   AI_710B.RAW_MIN := -2000;
   AI_710B.RAW_MAX := 8500;
   AI_710B.RAW_NAME := 'Thermal Resistance - 4-wire (Pt200 standard - 3916)';
   AI_710B.___________0030_1 := false;
   AI_710B.___________0030_2 := false;
   AI_710B.PARAM_TYPE := 16#07;
   AI_710B.PARAM_RANGE := 16#0B;
   AI_710B.PARAM_COEF := 16#01;
   AI_710B.VALUE_COEF := 0.003916;
   AI_730B.AI_CODE := 16#730B;
   AI_730B.___________0020_0 := false;
   AI_730B.___________0010_2 := false;
   AI_730B.RAW_MIN := -2000;
   AI_730B.RAW_MAX := 8500;
   AI_730B.RAW_NAME := 'Thermal Resistance - 4-wire (Pt200 standard - 392)';
   AI_730B.___________0030_1 := false;
   AI_730B.___________0030_2 := false;
   AI_730B.PARAM_TYPE := 16#07;
   AI_730B.PARAM_RANGE := 16#0B;
   AI_730B.PARAM_COEF := 16#03;
   AI_730B.VALUE_COEF := 0.00392;
   AI_7008.AI_CODE := 16#7008;
   AI_7008.___________0020_0 := false;
   AI_7008.___________0010_2 := false;
   AI_7008.RAW_MIN := -12000;
   AI_7008.RAW_MAX := 13000;
   AI_7008.RAW_NAME := 'Thermal Resistance - 4-wire (Pt500 climate - 3851)';
   AI_7008.___________0030_1 := false;
   AI_7008.___________0030_2 := false;
   AI_7008.PARAM_TYPE := 16#07;
   AI_7008.PARAM_RANGE := 16#08;
   AI_7008.PARAM_COEF := 16#00;
   AI_7008.VALUE_COEF := 0.003851;
   AI_7208.AI_CODE := 16#7208;
   AI_7208.___________0020_0 := false;
   AI_7208.___________0010_2 := false;
   AI_7208.RAW_MIN := -12000;
   AI_7208.RAW_MAX := 13000;
   AI_7208.RAW_NAME := 'Thermal Resistance - 4-wire (Pt500 climate - 3902)';
   AI_7208.___________0030_1 := false;
   AI_7208.___________0030_2 := false;
   AI_7208.PARAM_TYPE := 16#07;
   AI_7208.PARAM_RANGE := 16#08;
   AI_7208.PARAM_COEF := 16#02;
   AI_7208.VALUE_COEF := 0.003902;
   AI_7508.AI_CODE := 16#7508;
   AI_7508.___________0020_0 := false;
   AI_7508.___________0010_2 := false;
   AI_7508.RAW_MIN := -12000;
   AI_7508.RAW_MAX := 13000;
   AI_7508.RAW_NAME := 'Thermal Resistance - 4-wire (Pt500 climate - 391)';
   AI_7508.___________0030_1 := false;
   AI_7508.___________0030_2 := false;
   AI_7508.PARAM_TYPE := 16#07;
   AI_7508.PARAM_RANGE := 16#08;
   AI_7508.PARAM_COEF := 16#05;
   AI_7508.VALUE_COEF := 0.00391;
   AI_7108.AI_CODE := 16#7108;
   AI_7108.___________0020_0 := false;
   AI_7108.___________0010_2 := false;
   AI_7108.RAW_MIN := -12000;
   AI_7108.RAW_MAX := 13000;
   AI_7108.RAW_NAME := 'Thermal Resistance - 4-wire (Pt500 climate - 3916)';
   AI_7108.___________0030_1 := false;
   AI_7108.___________0030_2 := false;
   AI_7108.PARAM_TYPE := 16#07;
   AI_7108.PARAM_RANGE := 16#08;
   AI_7108.PARAM_COEF := 16#01;
   AI_7108.VALUE_COEF := 0.003916;
   AI_7308.AI_CODE := 16#7308;
   AI_7308.___________0020_0 := false;
   AI_7308.___________0010_2 := false;
   AI_7308.RAW_MIN := -12000;
   AI_7308.RAW_MAX := 13000;
   AI_7308.RAW_NAME := 'Thermal Resistance - 4-wire (Pt500 climate - 392)';
   AI_7308.___________0030_1 := false;
   AI_7308.___________0030_2 := false;
   AI_7308.PARAM_TYPE := 16#07;
   AI_7308.PARAM_RANGE := 16#08;
   AI_7308.PARAM_COEF := 16#03;
   AI_7308.VALUE_COEF := 0.00392;
   AI_7004.AI_CODE := 16#7004;
   AI_7004.___________0020_0 := false;
   AI_7004.___________0010_2 := false;
   AI_7004.RAW_MIN := -2000;
   AI_7004.RAW_MAX := 8500;
   AI_7004.RAW_NAME := 'Thermal Resistance - 4-wire (Pt500 standard - 3851)';
   AI_7004.___________0030_1 := false;
   AI_7004.___________0030_2 := false;
   AI_7004.PARAM_TYPE := 16#07;
   AI_7004.PARAM_RANGE := 16#04;
   AI_7004.PARAM_COEF := 16#00;
   AI_7004.VALUE_COEF := 0.003851;
   AI_7204.AI_CODE := 16#7204;
   AI_7204.___________0020_0 := false;
   AI_7204.___________0010_2 := false;
   AI_7204.RAW_MIN := -2000;
   AI_7204.RAW_MAX := 8500;
   AI_7204.RAW_NAME := 'Thermal Resistance - 4-wire (Pt500 standard - 3902)';
   AI_7204.___________0030_1 := false;
   AI_7204.___________0030_2 := false;
   AI_7204.PARAM_TYPE := 16#07;
   AI_7204.PARAM_RANGE := 16#04;
   AI_7204.PARAM_COEF := 16#02;
   AI_7204.VALUE_COEF := 0.003902;
   AI_7504.AI_CODE := 16#7504;
   AI_7504.___________0020_0 := false;
   AI_7504.___________0010_2 := false;
   AI_7504.RAW_MIN := -2000;
   AI_7504.RAW_MAX := 8500;
   AI_7504.RAW_NAME := 'Thermal Resistance - 4-wire (Pt500 standard - 391)';
   AI_7504.___________0030_1 := false;
   AI_7504.___________0030_2 := false;
   AI_7504.PARAM_TYPE := 16#07;
   AI_7504.PARAM_RANGE := 16#04;
   AI_7504.PARAM_COEF := 16#05;
   AI_7504.VALUE_COEF := 0.00391;
   AI_7104.AI_CODE := 16#7104;
   AI_7104.___________0020_0 := false;
   AI_7104.___________0010_2 := false;
   AI_7104.RAW_MIN := -2000;
   AI_7104.RAW_MAX := 8500;
   AI_7104.RAW_NAME := 'Thermal Resistance - 4-wire (Pt500 standard - 3916)';
   AI_7104.___________0030_1 := false;
   AI_7104.___________0030_2 := false;
   AI_7104.PARAM_TYPE := 16#07;
   AI_7104.PARAM_RANGE := 16#04;
   AI_7104.PARAM_COEF := 16#01;
   AI_7104.VALUE_COEF := 0.003916;
   AI_7304.AI_CODE := 16#7304;
   AI_7304.___________0020_0 := false;
   AI_7304.___________0010_2 := false;
   AI_7304.RAW_MIN := -2000;
   AI_7304.RAW_MAX := 8500;
   AI_7304.RAW_NAME := 'Thermal Resistance - 4-wire (Pt500 standard - 392)';
   AI_7304.___________0030_1 := false;
   AI_7304.___________0030_2 := false;
   AI_7304.PARAM_TYPE := 16#07;
   AI_7304.PARAM_RANGE := 16#04;
   AI_7304.PARAM_COEF := 16#03;
   AI_7304.VALUE_COEF := 0.00392;
   AI_7009.AI_CODE := 16#7009;
   AI_7009.___________0020_0 := false;
   AI_7009.___________0010_2 := false;
   AI_7009.RAW_MIN := -12000;
   AI_7009.RAW_MAX := 13000;
   AI_7009.RAW_NAME := 'Thermal Resistance - 4-wire (Pt1000 climate - 3851)';
   AI_7009.___________0030_1 := false;
   AI_7009.___________0030_2 := false;
   AI_7009.PARAM_TYPE := 16#07;
   AI_7009.PARAM_RANGE := 16#09;
   AI_7009.PARAM_COEF := 16#00;
   AI_7009.VALUE_COEF := 0.003851;
   AI_7209.AI_CODE := 16#7209;
   AI_7209.___________0020_0 := false;
   AI_7209.___________0010_2 := false;
   AI_7209.RAW_MIN := -12000;
   AI_7209.RAW_MAX := 13000;
   AI_7209.RAW_NAME := 'Thermal Resistance - 4-wire (Pt1000 climate - 3902)';
   AI_7209.___________0030_1 := false;
   AI_7209.___________0030_2 := false;
   AI_7209.PARAM_TYPE := 16#07;
   AI_7209.PARAM_RANGE := 16#09;
   AI_7209.PARAM_COEF := 16#02;
   AI_7209.VALUE_COEF := 0.003902;
   AI_7509.AI_CODE := 16#7509;
   AI_7509.___________0020_0 := false;
   AI_7509.___________0010_2 := false;
   AI_7509.RAW_MIN := -12000;
   AI_7509.RAW_MAX := 13000;
   AI_7509.RAW_NAME := 'Thermal Resistance - 4-wire (Pt1000 climate - 391)';
   AI_7509.___________0030_1 := false;
   AI_7509.___________0030_2 := false;
   AI_7509.PARAM_TYPE := 16#07;
   AI_7509.PARAM_RANGE := 16#09;
   AI_7509.PARAM_COEF := 16#05;
   AI_7509.VALUE_COEF := 0.00391;
   AI_7109.AI_CODE := 16#7109;
   AI_7109.___________0020_0 := false;
   AI_7109.___________0010_2 := false;
   AI_7109.RAW_MIN := -12000;
   AI_7109.RAW_MAX := 13000;
   AI_7109.RAW_NAME := 'Thermal Resistance - 4-wire (Pt1000 climate - 3916)';
   AI_7109.___________0030_1 := false;
   AI_7109.___________0030_2 := false;
   AI_7109.PARAM_TYPE := 16#07;
   AI_7109.PARAM_RANGE := 16#09;
   AI_7109.PARAM_COEF := 16#01;
   AI_7109.VALUE_COEF := 0.003916;
   AI_7309.AI_CODE := 16#7309;
   AI_7309.___________0020_0 := false;
   AI_7309.___________0010_2 := false;
   AI_7309.RAW_MIN := -12000;
   AI_7309.RAW_MAX := 13000;
   AI_7309.RAW_NAME := 'Thermal Resistance - 4-wire (Pt1000 climate - 392)';
   AI_7309.___________0030_1 := false;
   AI_7309.___________0030_2 := false;
   AI_7309.PARAM_TYPE := 16#07;
   AI_7309.PARAM_RANGE := 16#09;
   AI_7309.PARAM_COEF := 16#03;
   AI_7309.VALUE_COEF := 0.00392;
   AI_7005.AI_CODE := 16#7005;
   AI_7005.___________0020_0 := false;
   AI_7005.___________0010_2 := false;
   AI_7005.RAW_MIN := -2000;
   AI_7005.RAW_MAX := 8500;
   AI_7005.RAW_NAME := 'Thermal Resistance - 4-wire (Pt1000 standard - 3851)';
   AI_7005.___________0030_1 := false;
   AI_7005.___________0030_2 := false;
   AI_7005.PARAM_TYPE := 16#07;
   AI_7005.PARAM_RANGE := 16#05;
   AI_7005.PARAM_COEF := 16#00;
   AI_7005.VALUE_COEF := 0.003851;
   AI_7205.AI_CODE := 16#7205;
   AI_7205.___________0020_0 := false;
   AI_7205.___________0010_2 := false;
   AI_7205.RAW_MIN := -2000;
   AI_7205.RAW_MAX := 8500;
   AI_7205.RAW_NAME := 'Thermal Resistance - 4-wire (Pt1000 standard - 3902)';
   AI_7205.___________0030_1 := false;
   AI_7205.___________0030_2 := false;
   AI_7205.PARAM_TYPE := 16#07;
   AI_7205.PARAM_RANGE := 16#05;
   AI_7205.PARAM_COEF := 16#02;
   AI_7205.VALUE_COEF := 0.003902;
   AI_7505.AI_CODE := 16#7505;
   AI_7505.___________0020_0 := false;
   AI_7505.___________0010_2 := false;
   AI_7505.RAW_MIN := -2000;
   AI_7505.RAW_MAX := 8500;
   AI_7505.RAW_NAME := 'Thermal Resistance - 4-wire (Pt1000 standard - 391)';
   AI_7505.___________0030_1 := false;
   AI_7505.___________0030_2 := false;
   AI_7505.PARAM_TYPE := 16#07;
   AI_7505.PARAM_RANGE := 16#05;
   AI_7505.PARAM_COEF := 16#05;
   AI_7505.VALUE_COEF := 0.00391;
   AI_7105.AI_CODE := 16#7105;
   AI_7105.___________0020_0 := false;
   AI_7105.___________0010_2 := false;
   AI_7105.RAW_MIN := -2000;
   AI_7105.RAW_MAX := 8500;
   AI_7105.RAW_NAME := 'Thermal Resistance - 4-wire (Pt1000 standard - 3916)';
   AI_7105.___________0030_1 := false;
   AI_7105.___________0030_2 := false;
   AI_7105.PARAM_TYPE := 16#07;
   AI_7105.PARAM_RANGE := 16#05;
   AI_7105.PARAM_COEF := 16#01;
   AI_7105.VALUE_COEF := 0.003916;
   AI_7305.AI_CODE := 16#7305;
   AI_7305.___________0020_0 := false;
   AI_7305.___________0010_2 := false;
   AI_7305.RAW_MIN := -2000;
   AI_7305.RAW_MAX := 8500;
   AI_7305.RAW_NAME := 'Thermal Resistance - 4-wire (Pt1000 standard - 392)';
   AI_7305.___________0030_1 := false;
   AI_7305.___________0030_2 := false;
   AI_7305.PARAM_TYPE := 16#07;
   AI_7305.PARAM_RANGE := 16#05;
   AI_7305.PARAM_COEF := 16#03;
   AI_7305.VALUE_COEF := 0.00392;
   AI_8B0E.AI_CODE := 16#8B0E;
   AI_8B0E.___________0020_0 := false;
   AI_8B0E.___________0010_2 := false;
   AI_8B0E.RAW_MIN := -5000;
   AI_8B0E.RAW_MAX := 15000;
   AI_8B0E.RAW_NAME := 'Thermal Resistance - 3-wire (Cu10 climate - 426)';
   AI_8B0E.___________0030_1 := false;
   AI_8B0E.___________0030_2 := false;
   AI_8B0E.PARAM_TYPE := 16#08;
   AI_8B0E.PARAM_RANGE := 16#0E;
   AI_8B0E.PARAM_COEF := 16#0B;
   AI_8B0E.VALUE_COEF := 0.00426;
   AI_8C0E.AI_CODE := 16#8C0E;
   AI_8C0E.___________0020_0 := false;
   AI_8C0E.___________0010_2 := false;
   AI_8C0E.RAW_MIN := -5000;
   AI_8C0E.RAW_MAX := 15000;
   AI_8C0E.RAW_NAME := 'Thermal Resistance - 3-wire (Cu10 climate - 427)';
   AI_8C0E.___________0030_1 := false;
   AI_8C0E.___________0030_2 := false;
   AI_8C0E.PARAM_TYPE := 16#08;
   AI_8C0E.PARAM_RANGE := 16#0E;
   AI_8C0E.PARAM_COEF := 16#0C;
   AI_8C0E.VALUE_COEF := 0.00427;
   AI_8D0E.AI_CODE := 16#8D0E;
   AI_8D0E.___________0020_0 := false;
   AI_8D0E.___________0010_2 := false;
   AI_8D0E.RAW_MIN := -5000;
   AI_8D0E.RAW_MAX := 15000;
   AI_8D0E.RAW_NAME := 'Thermal Resistance - 3-wire (Cu10 climate - 428)';
   AI_8D0E.___________0030_1 := false;
   AI_8D0E.___________0030_2 := false;
   AI_8D0E.PARAM_TYPE := 16#08;
   AI_8D0E.PARAM_RANGE := 16#0E;
   AI_8D0E.PARAM_COEF := 16#0D;
   AI_8D0E.VALUE_COEF := 0.00428;
   AI_8B0F.AI_CODE := 16#8B0F;
   AI_8B0F.___________0020_0 := false;
   AI_8B0F.___________0010_2 := false;
   AI_8B0F.RAW_MIN := -500;
   AI_8B0F.RAW_MAX := 2000;
   AI_8B0F.RAW_NAME := 'Thermal Resistance - 3-wire (Cu10 standard - 426)';
   AI_8B0F.___________0030_1 := false;
   AI_8B0F.___________0030_2 := false;
   AI_8B0F.PARAM_TYPE := 16#08;
   AI_8B0F.PARAM_RANGE := 16#0F;
   AI_8B0F.PARAM_COEF := 16#0B;
   AI_8B0F.VALUE_COEF := 0.00426;
   AI_8C0F.AI_CODE := 16#8C0F;
   AI_8C0F.___________0020_0 := false;
   AI_8C0F.___________0010_2 := false;
   AI_8C0F.RAW_MIN := -2000;
   AI_8C0F.RAW_MAX := 2600;
   AI_8C0F.RAW_NAME := 'Thermal Resistance - 3-wire (Cu10 standard - 427)';
   AI_8C0F.___________0030_1 := false;
   AI_8C0F.___________0030_2 := false;
   AI_8C0F.PARAM_TYPE := 16#08;
   AI_8C0F.PARAM_RANGE := 16#0F;
   AI_8C0F.PARAM_COEF := 16#0C;
   AI_8C0F.VALUE_COEF := 0.00427;
   AI_8D0F.AI_CODE := 16#8D0F;
   AI_8D0F.___________0020_0 := false;
   AI_8D0F.___________0010_2 := false;
   AI_8D0F.RAW_MIN := -1800;
   AI_8D0F.RAW_MAX := 2000;
   AI_8D0F.RAW_NAME := 'Thermal Resistance - 3-wire (Cu10 standard - 428)';
   AI_8D0F.___________0030_1 := false;
   AI_8D0F.___________0030_2 := false;
   AI_8D0F.PARAM_TYPE := 16#08;
   AI_8D0F.PARAM_RANGE := 16#0F;
   AI_8D0F.PARAM_COEF := 16#0D;
   AI_8D0F.VALUE_COEF := 0.00428;
   AI_8B19.AI_CODE := 16#8B19;
   AI_8B19.___________0020_0 := false;
   AI_8B19.___________0010_2 := false;
   AI_8B19.RAW_MIN := -5000;
   AI_8B19.RAW_MAX := 15000;
   AI_8B19.RAW_NAME := 'Thermal Resistance - 3-wire (Cu50 climate - 426)';
   AI_8B19.___________0030_1 := false;
   AI_8B19.___________0030_2 := false;
   AI_8B19.PARAM_TYPE := 16#08;
   AI_8B19.PARAM_RANGE := 16#19;
   AI_8B19.PARAM_COEF := 16#0B;
   AI_8B19.VALUE_COEF := 0.00426;
   AI_8C19.AI_CODE := 16#8C19;
   AI_8C19.___________0020_0 := false;
   AI_8C19.___________0010_2 := false;
   AI_8C19.RAW_MIN := -5000;
   AI_8C19.RAW_MAX := 15000;
   AI_8C19.RAW_NAME := 'Thermal Resistance - 3-wire (Cu50 climate - 427)';
   AI_8C19.___________0030_1 := false;
   AI_8C19.___________0030_2 := false;
   AI_8C19.PARAM_TYPE := 16#08;
   AI_8C19.PARAM_RANGE := 16#19;
   AI_8C19.PARAM_COEF := 16#0C;
   AI_8C19.VALUE_COEF := 0.00427;
   AI_8D19.AI_CODE := 16#8D19;
   AI_8D19.___________0020_0 := false;
   AI_8D19.___________0010_2 := false;
   AI_8D19.RAW_MIN := -5000;
   AI_8D19.RAW_MAX := 15000;
   AI_8D19.RAW_NAME := 'Thermal Resistance - 3-wire (Cu50 climate - 428)';
   AI_8D19.___________0030_1 := false;
   AI_8D19.___________0030_2 := false;
   AI_8D19.PARAM_TYPE := 16#08;
   AI_8D19.PARAM_RANGE := 16#19;
   AI_8D19.PARAM_COEF := 16#0D;
   AI_8D19.VALUE_COEF := 0.00428;
   AI_8B18.AI_CODE := 16#8B18;
   AI_8B18.___________0020_0 := false;
   AI_8B18.___________0010_2 := false;
   AI_8B18.RAW_MIN := -500;
   AI_8B18.RAW_MAX := 2000;
   AI_8B18.RAW_NAME := 'Thermal Resistance - 3-wire (Cu50 standard - 426)';
   AI_8B18.___________0030_1 := false;
   AI_8B18.___________0030_2 := false;
   AI_8B18.PARAM_TYPE := 16#08;
   AI_8B18.PARAM_RANGE := 16#18;
   AI_8B18.PARAM_COEF := 16#0B;
   AI_8B18.VALUE_COEF := 0.00426;
   AI_8C18.AI_CODE := 16#8C18;
   AI_8C18.___________0020_0 := false;
   AI_8C18.___________0010_2 := false;
   AI_8C18.RAW_MIN := -2000;
   AI_8C18.RAW_MAX := 2600;
   AI_8C18.RAW_NAME := 'Thermal Resistance - 3-wire (Cu50 standard - 427)';
   AI_8C18.___________0030_1 := false;
   AI_8C18.___________0030_2 := false;
   AI_8C18.PARAM_TYPE := 16#08;
   AI_8C18.PARAM_RANGE := 16#18;
   AI_8C18.PARAM_COEF := 16#0C;
   AI_8C18.VALUE_COEF := 0.00427;
   AI_8D18.AI_CODE := 16#8D18;
   AI_8D18.___________0020_0 := false;
   AI_8D18.___________0010_2 := false;
   AI_8D18.RAW_MIN := -1800;
   AI_8D18.RAW_MAX := 2000;
   AI_8D18.RAW_NAME := 'Thermal Resistance - 3-wire (Cu50 standard - 428)';
   AI_8D18.___________0030_1 := false;
   AI_8D18.___________0030_2 := false;
   AI_8D18.PARAM_TYPE := 16#08;
   AI_8D18.PARAM_RANGE := 16#18;
   AI_8D18.PARAM_COEF := 16#0D;
   AI_8D18.VALUE_COEF := 0.00428;
   AI_8B1B.AI_CODE := 16#8B1B;
   AI_8B1B.___________0020_0 := false;
   AI_8B1B.___________0010_2 := false;
   AI_8B1B.RAW_MIN := -5000;
   AI_8B1B.RAW_MAX := 15000;
   AI_8B1B.RAW_NAME := 'Thermal Resistance - 3-wire (Cu100 climate - 426)';
   AI_8B1B.___________0030_1 := false;
   AI_8B1B.___________0030_2 := false;
   AI_8B1B.PARAM_TYPE := 16#08;
   AI_8B1B.PARAM_RANGE := 16#1B;
   AI_8B1B.PARAM_COEF := 16#0B;
   AI_8B1B.VALUE_COEF := 0.00426;
   AI_8C1B.AI_CODE := 16#8C1B;
   AI_8C1B.___________0020_0 := false;
   AI_8C1B.___________0010_2 := false;
   AI_8C1B.RAW_MIN := -5000;
   AI_8C1B.RAW_MAX := 15000;
   AI_8C1B.RAW_NAME := 'Thermal Resistance - 3-wire (Cu100 climate - 427)';
   AI_8C1B.___________0030_1 := false;
   AI_8C1B.___________0030_2 := false;
   AI_8C1B.PARAM_TYPE := 16#08;
   AI_8C1B.PARAM_RANGE := 16#1B;
   AI_8C1B.PARAM_COEF := 16#0C;
   AI_8C1B.VALUE_COEF := 0.00427;
   AI_8D1B.AI_CODE := 16#8D1B;
   AI_8D1B.___________0020_0 := false;
   AI_8D1B.___________0010_2 := false;
   AI_8D1B.RAW_MIN := -5000;
   AI_8D1B.RAW_MAX := 15000;
   AI_8D1B.RAW_NAME := 'Thermal Resistance - 3-wire (Cu100 climate - 428)';
   AI_8D1B.___________0030_1 := false;
   AI_8D1B.___________0030_2 := false;
   AI_8D1B.PARAM_TYPE := 16#08;
   AI_8D1B.PARAM_RANGE := 16#1B;
   AI_8D1B.PARAM_COEF := 16#0D;
   AI_8D1B.VALUE_COEF := 0.00428;
   AI_8B1A.AI_CODE := 16#8B1A;
   AI_8B1A.___________0020_0 := false;
   AI_8B1A.___________0010_2 := false;
   AI_8B1A.RAW_MIN := -500;
   AI_8B1A.RAW_MAX := 2000;
   AI_8B1A.RAW_NAME := 'Thermal Resistance - 3-wire (Cu100 standard - 426)';
   AI_8B1A.___________0030_1 := false;
   AI_8B1A.___________0030_2 := false;
   AI_8B1A.PARAM_TYPE := 16#08;
   AI_8B1A.PARAM_RANGE := 16#1A;
   AI_8B1A.PARAM_COEF := 16#0B;
   AI_8B1A.VALUE_COEF := 0.00426;
   AI_8C1A.AI_CODE := 16#8C1A;
   AI_8C1A.___________0020_0 := false;
   AI_8C1A.___________0010_2 := false;
   AI_8C1A.RAW_MIN := -2000;
   AI_8C1A.RAW_MAX := 2600;
   AI_8C1A.RAW_NAME := 'Thermal Resistance - 3-wire (Cu100 standard - 427)';
   AI_8C1A.___________0030_1 := false;
   AI_8C1A.___________0030_2 := false;
   AI_8C1A.PARAM_TYPE := 16#08;
   AI_8C1A.PARAM_RANGE := 16#1A;
   AI_8C1A.PARAM_COEF := 16#0C;
   AI_8C1A.VALUE_COEF := 0.00427;
   AI_8D1A.AI_CODE := 16#8D1A;
   AI_8D1A.___________0020_0 := false;
   AI_8D1A.___________0010_2 := false;
   AI_8D1A.RAW_MIN := -1800;
   AI_8D1A.RAW_MAX := 2000;
   AI_8D1A.RAW_NAME := 'Thermal Resistance - 3-wire (Cu100 standard - 428)';
   AI_8D1A.___________0030_1 := false;
   AI_8D1A.___________0030_2 := false;
   AI_8D1A.PARAM_TYPE := 16#08;
   AI_8D1A.PARAM_RANGE := 16#1A;
   AI_8D1A.PARAM_COEF := 16#0D;
   AI_8D1A.VALUE_COEF := 0.00428;
   AI_8A1D.AI_CODE := 16#8A1D;
   AI_8A1D.___________0020_0 := false;
   AI_8A1D.___________0010_2 := false;
   AI_8A1D.RAW_MIN := -6000;
   AI_8A1D.RAW_MAX := 13000;
   AI_8A1D.RAW_NAME := 'Thermal Resistance - 3-wire (LG-Ni1000 climate - 500)';
   AI_8A1D.___________0030_1 := false;
   AI_8A1D.___________0030_2 := false;
   AI_8A1D.PARAM_TYPE := 16#08;
   AI_8A1D.PARAM_RANGE := 16#1D;
   AI_8A1D.PARAM_COEF := 16#0A;
   AI_8A1D.VALUE_COEF := 0.005;
   AI_8A1C.AI_CODE := 16#8A1C;
   AI_8A1C.___________0020_0 := false;
   AI_8A1C.___________0010_2 := false;
   AI_8A1C.RAW_MIN := -600;
   AI_8A1C.RAW_MAX := 2500;
   AI_8A1C.RAW_NAME := 'Thermal Resistance - 3-wire (LG-Ni1000 standard - 500)';
   AI_8A1C.___________0030_1 := false;
   AI_8A1C.___________0030_2 := false;
   AI_8A1C.PARAM_TYPE := 16#08;
   AI_8A1C.PARAM_RANGE := 16#1C;
   AI_8A1C.PARAM_COEF := 16#0A;
   AI_8A1C.VALUE_COEF := 0.005;
   AI_871F.AI_CODE := 16#871F;
   AI_871F.___________0020_0 := false;
   AI_871F.___________0010_2 := false;
   AI_871F.RAW_MIN := -6000;
   AI_871F.RAW_MAX := 13000;
   AI_871F.RAW_NAME := 'Thermal Resistance - 3-wire (Ni10 climate - 617)';
   AI_871F.___________0030_1 := false;
   AI_871F.___________0030_2 := false;
   AI_871F.PARAM_TYPE := 16#08;
   AI_871F.PARAM_RANGE := 16#1F;
   AI_871F.PARAM_COEF := 16#07;
   AI_871F.VALUE_COEF := 0.00617;
   AI_881F.AI_CODE := 16#881F;
   AI_881F.___________0020_0 := false;
   AI_881F.___________0010_2 := false;
   AI_881F.RAW_MIN := -6000;
   AI_881F.RAW_MAX := 13000;
   AI_881F.RAW_NAME := 'Thermal Resistance - 3-wire (Ni10 climate - 618)';
   AI_881F.___________0030_1 := false;
   AI_881F.___________0030_2 := false;
   AI_881F.PARAM_TYPE := 16#08;
   AI_881F.PARAM_RANGE := 16#1F;
   AI_881F.PARAM_COEF := 16#08;
   AI_881F.VALUE_COEF := 0.00618;
   AI_891F.AI_CODE := 16#891F;
   AI_891F.___________0020_0 := false;
   AI_891F.___________0010_2 := false;
   AI_891F.RAW_MIN := -6000;
   AI_891F.RAW_MAX := 13000;
   AI_891F.RAW_NAME := 'Thermal Resistance - 3-wire (Ni10 climate - 672)';
   AI_891F.___________0030_1 := false;
   AI_891F.___________0030_2 := false;
   AI_891F.PARAM_TYPE := 16#08;
   AI_891F.PARAM_RANGE := 16#1F;
   AI_891F.PARAM_COEF := 16#09;
   AI_891F.VALUE_COEF := 0.00672;
   AI_871E.AI_CODE := 16#871E;
   AI_871E.___________0020_0 := false;
   AI_871E.___________0010_2 := false;
   AI_871E.RAW_MIN := -600;
   AI_871E.RAW_MAX := 1800;
   AI_871E.RAW_NAME := 'Thermal Resistance - 3-wire (Ni10 standard - 617)';
   AI_871E.___________0030_1 := false;
   AI_871E.___________0030_2 := false;
   AI_871E.PARAM_TYPE := 16#08;
   AI_871E.PARAM_RANGE := 16#1E;
   AI_871E.PARAM_COEF := 16#07;
   AI_871E.VALUE_COEF := 0.00617;
   AI_881E.AI_CODE := 16#881E;
   AI_881E.___________0020_0 := false;
   AI_881E.___________0010_2 := false;
   AI_881E.RAW_MIN := -600;
   AI_881E.RAW_MAX := 2500;
   AI_881E.RAW_NAME := 'Thermal Resistance - 3-wire (Ni10 standard - 618)';
   AI_881E.___________0030_1 := false;
   AI_881E.___________0030_2 := false;
   AI_881E.PARAM_TYPE := 16#08;
   AI_881E.PARAM_RANGE := 16#1E;
   AI_881E.PARAM_COEF := 16#08;
   AI_881E.VALUE_COEF := 0.00618;
   AI_891E.AI_CODE := 16#891E;
   AI_891E.___________0020_0 := false;
   AI_891E.___________0010_2 := false;
   AI_891E.RAW_MIN := -600;
   AI_891E.RAW_MAX := 2500;
   AI_891E.RAW_NAME := 'Thermal Resistance - 3-wire (Ni10 standard - 672)';
   AI_891E.___________0030_1 := false;
   AI_891E.___________0030_2 := false;
   AI_891E.PARAM_TYPE := 16#08;
   AI_891E.PARAM_RANGE := 16#1E;
   AI_891E.PARAM_COEF := 16#09;
   AI_891E.VALUE_COEF := 0.00672;
   AI_870D.AI_CODE := 16#870D;
   AI_870D.___________0020_0 := false;
   AI_870D.___________0010_2 := false;
   AI_870D.RAW_MIN := -6000;
   AI_870D.RAW_MAX := 13000;
   AI_870D.RAW_NAME := 'Thermal Resistance - 3-wire (Ni120 climate - 617)';
   AI_870D.___________0030_1 := false;
   AI_870D.___________0030_2 := false;
   AI_870D.PARAM_TYPE := 16#08;
   AI_870D.PARAM_RANGE := 16#0D;
   AI_870D.PARAM_COEF := 16#07;
   AI_870D.VALUE_COEF := 0.00617;
   AI_880D.AI_CODE := 16#880D;
   AI_880D.___________0020_0 := false;
   AI_880D.___________0010_2 := false;
   AI_880D.RAW_MIN := -6000;
   AI_880D.RAW_MAX := 13000;
   AI_880D.RAW_NAME := 'Thermal Resistance - 3-wire (Ni120 climate - 618)';
   AI_880D.___________0030_1 := false;
   AI_880D.___________0030_2 := false;
   AI_880D.PARAM_TYPE := 16#08;
   AI_880D.PARAM_RANGE := 16#0D;
   AI_880D.PARAM_COEF := 16#08;
   AI_880D.VALUE_COEF := 0.00618;
   AI_890D.AI_CODE := 16#890D;
   AI_890D.___________0020_0 := false;
   AI_890D.___________0010_2 := false;
   AI_890D.RAW_MIN := -6000;
   AI_890D.RAW_MAX := 13000;
   AI_890D.RAW_NAME := 'Thermal Resistance - 3-wire (Ni120 climate - 672)';
   AI_890D.___________0030_1 := false;
   AI_890D.___________0030_2 := false;
   AI_890D.PARAM_TYPE := 16#08;
   AI_890D.PARAM_RANGE := 16#0D;
   AI_890D.PARAM_COEF := 16#09;
   AI_890D.VALUE_COEF := 0.00672;
   AI_870C.AI_CODE := 16#870C;
   AI_870C.___________0020_0 := false;
   AI_870C.___________0010_2 := false;
   AI_870C.RAW_MIN := -600;
   AI_870C.RAW_MAX := 1800;
   AI_870C.RAW_NAME := 'Thermal Resistance - 3-wire (Ni120 standard - 617)';
   AI_870C.___________0030_1 := false;
   AI_870C.___________0030_2 := false;
   AI_870C.PARAM_TYPE := 16#08;
   AI_870C.PARAM_RANGE := 16#0C;
   AI_870C.PARAM_COEF := 16#07;
   AI_870C.VALUE_COEF := 0.00617;
   AI_880C.AI_CODE := 16#880C;
   AI_880C.___________0020_0 := false;
   AI_880C.___________0010_2 := false;
   AI_880C.RAW_MIN := -600;
   AI_880C.RAW_MAX := 2500;
   AI_880C.RAW_NAME := 'Thermal Resistance - 3-wire (Ni120 standard - 618)';
   AI_880C.___________0030_1 := false;
   AI_880C.___________0030_2 := false;
   AI_880C.PARAM_TYPE := 16#08;
   AI_880C.PARAM_RANGE := 16#0C;
   AI_880C.PARAM_COEF := 16#08;
   AI_880C.VALUE_COEF := 0.00618;
   AI_890C.AI_CODE := 16#890C;
   AI_890C.___________0020_0 := false;
   AI_890C.___________0010_2 := false;
   AI_890C.RAW_MIN := -600;
   AI_890C.RAW_MAX := 2500;
   AI_890C.RAW_NAME := 'Thermal Resistance - 3-wire (Ni120 standard - 672)';
   AI_890C.___________0030_1 := false;
   AI_890C.___________0030_2 := false;
   AI_890C.PARAM_TYPE := 16#08;
   AI_890C.PARAM_RANGE := 16#0C;
   AI_890C.PARAM_COEF := 16#09;
   AI_890C.VALUE_COEF := 0.00672;
   AI_8701.AI_CODE := 16#8701;
   AI_8701.___________0020_0 := false;
   AI_8701.___________0010_2 := false;
   AI_8701.RAW_MIN := -6000;
   AI_8701.RAW_MAX := 13000;
   AI_8701.RAW_NAME := 'Thermal Resistance - 3-wire (Ni100 climate - 617)';
   AI_8701.___________0030_1 := false;
   AI_8701.___________0030_2 := false;
   AI_8701.PARAM_TYPE := 16#08;
   AI_8701.PARAM_RANGE := 16#01;
   AI_8701.PARAM_COEF := 16#07;
   AI_8701.VALUE_COEF := 0.00617;
   AI_8801.AI_CODE := 16#8801;
   AI_8801.___________0020_0 := false;
   AI_8801.___________0010_2 := false;
   AI_8801.RAW_MIN := -6000;
   AI_8801.RAW_MAX := 13000;
   AI_8801.RAW_NAME := 'Thermal Resistance - 3-wire (Ni100 climate - 618)';
   AI_8801.___________0030_1 := false;
   AI_8801.___________0030_2 := false;
   AI_8801.PARAM_TYPE := 16#08;
   AI_8801.PARAM_RANGE := 16#01;
   AI_8801.PARAM_COEF := 16#08;
   AI_8801.VALUE_COEF := 0.00618;
   AI_8901.AI_CODE := 16#8901;
   AI_8901.___________0020_0 := false;
   AI_8901.___________0010_2 := false;
   AI_8901.RAW_MIN := -6000;
   AI_8901.RAW_MAX := 13000;
   AI_8901.RAW_NAME := 'Thermal Resistance - 3-wire (Ni100 climate - 672)';
   AI_8901.___________0030_1 := false;
   AI_8901.___________0030_2 := false;
   AI_8901.PARAM_TYPE := 16#08;
   AI_8901.PARAM_RANGE := 16#01;
   AI_8901.PARAM_COEF := 16#09;
   AI_8901.VALUE_COEF := 0.00672;
   AI_8703.AI_CODE := 16#8703;
   AI_8703.___________0020_0 := false;
   AI_8703.___________0010_2 := false;
   AI_8703.RAW_MIN := -600;
   AI_8703.RAW_MAX := 1800;
   AI_8703.RAW_NAME := 'Thermal Resistance - 3-wire (Ni100 standard - 617)';
   AI_8703.___________0030_1 := false;
   AI_8703.___________0030_2 := false;
   AI_8703.PARAM_TYPE := 16#08;
   AI_8703.PARAM_RANGE := 16#03;
   AI_8703.PARAM_COEF := 16#07;
   AI_8703.VALUE_COEF := 0.00617;
   AI_8803.AI_CODE := 16#8803;
   AI_8803.___________0020_0 := false;
   AI_8803.___________0010_2 := false;
   AI_8803.RAW_MIN := -600;
   AI_8803.RAW_MAX := 2500;
   AI_8803.RAW_NAME := 'Thermal Resistance - 3-wire (Ni100 standard - 618)';
   AI_8803.___________0030_1 := false;
   AI_8803.___________0030_2 := false;
   AI_8803.PARAM_TYPE := 16#08;
   AI_8803.PARAM_RANGE := 16#03;
   AI_8803.PARAM_COEF := 16#08;
   AI_8803.VALUE_COEF := 0.00618;
   AI_8903.AI_CODE := 16#8903;
   AI_8903.___________0020_0 := false;
   AI_8903.___________0010_2 := false;
   AI_8903.RAW_MIN := -600;
   AI_8903.RAW_MAX := 2500;
   AI_8903.RAW_NAME := 'Thermal Resistance - 3-wire (Ni100 standard - 672)';
   AI_8903.___________0030_1 := false;
   AI_8903.___________0030_2 := false;
   AI_8903.PARAM_TYPE := 16#08;
   AI_8903.PARAM_RANGE := 16#03;
   AI_8903.PARAM_COEF := 16#09;
   AI_8903.VALUE_COEF := 0.00672;
   AI_8711.AI_CODE := 16#8711;
   AI_8711.___________0020_0 := false;
   AI_8711.___________0010_2 := false;
   AI_8711.RAW_MIN := -6000;
   AI_8711.RAW_MAX := 13000;
   AI_8711.RAW_NAME := 'Thermal Resistance - 3-wire (Ni200 climate - 617)';
   AI_8711.___________0030_1 := false;
   AI_8711.___________0030_2 := false;
   AI_8711.PARAM_TYPE := 16#08;
   AI_8711.PARAM_RANGE := 16#11;
   AI_8711.PARAM_COEF := 16#07;
   AI_8711.VALUE_COEF := 0.00617;
   AI_8811.AI_CODE := 16#8811;
   AI_8811.___________0020_0 := false;
   AI_8811.___________0010_2 := false;
   AI_8811.RAW_MIN := -6000;
   AI_8811.RAW_MAX := 13000;
   AI_8811.RAW_NAME := 'Thermal Resistance - 3-wire (Ni200 climate - 618)';
   AI_8811.___________0030_1 := false;
   AI_8811.___________0030_2 := false;
   AI_8811.PARAM_TYPE := 16#08;
   AI_8811.PARAM_RANGE := 16#11;
   AI_8811.PARAM_COEF := 16#08;
   AI_8811.VALUE_COEF := 0.00618;
   AI_8911.AI_CODE := 16#8911;
   AI_8911.___________0020_0 := false;
   AI_8911.___________0010_2 := false;
   AI_8911.RAW_MIN := -6000;
   AI_8911.RAW_MAX := 13000;
   AI_8911.RAW_NAME := 'Thermal Resistance - 3-wire (Ni200 climate - 672)';
   AI_8911.___________0030_1 := false;
   AI_8911.___________0030_2 := false;
   AI_8911.PARAM_TYPE := 16#08;
   AI_8911.PARAM_RANGE := 16#11;
   AI_8911.PARAM_COEF := 16#09;
   AI_8911.VALUE_COEF := 0.00672;
   AI_8710.AI_CODE := 16#8710;
   AI_8710.___________0020_0 := false;
   AI_8710.___________0010_2 := false;
   AI_8710.RAW_MIN := -600;
   AI_8710.RAW_MAX := 1800;
   AI_8710.RAW_NAME := 'Thermal Resistance - 3-wire (Ni200 standard - 617)';
   AI_8710.___________0030_1 := false;
   AI_8710.___________0030_2 := false;
   AI_8710.PARAM_TYPE := 16#08;
   AI_8710.PARAM_RANGE := 16#10;
   AI_8710.PARAM_COEF := 16#07;
   AI_8710.VALUE_COEF := 0.00617;
   AI_8810.AI_CODE := 16#8810;
   AI_8810.___________0020_0 := false;
   AI_8810.___________0010_2 := false;
   AI_8810.RAW_MIN := -600;
   AI_8810.RAW_MAX := 2500;
   AI_8810.RAW_NAME := 'Thermal Resistance - 3-wire (Ni200 standard - 618)';
   AI_8810.___________0030_1 := false;
   AI_8810.___________0030_2 := false;
   AI_8810.PARAM_TYPE := 16#08;
   AI_8810.PARAM_RANGE := 16#10;
   AI_8810.PARAM_COEF := 16#08;
   AI_8810.VALUE_COEF := 0.00618;
   AI_8910.AI_CODE := 16#8910;
   AI_8910.___________0020_0 := false;
   AI_8910.___________0010_2 := false;
   AI_8910.RAW_MIN := -600;
   AI_8910.RAW_MAX := 2500;
   AI_8910.RAW_NAME := 'Thermal Resistance - 3-wire (Ni200 standard - 672)';
   AI_8910.___________0030_1 := false;
   AI_8910.___________0030_2 := false;
   AI_8910.PARAM_TYPE := 16#08;
   AI_8910.PARAM_RANGE := 16#10;
   AI_8910.PARAM_COEF := 16#09;
   AI_8910.VALUE_COEF := 0.00672;
   AI_8713.AI_CODE := 16#8713;
   AI_8713.___________0020_0 := false;
   AI_8713.___________0010_2 := false;
   AI_8713.RAW_MIN := -6000;
   AI_8713.RAW_MAX := 13000;
   AI_8713.RAW_NAME := 'Thermal Resistance - 3-wire (Ni500 climate - 617)';
   AI_8713.___________0030_1 := false;
   AI_8713.___________0030_2 := false;
   AI_8713.PARAM_TYPE := 16#08;
   AI_8713.PARAM_RANGE := 16#13;
   AI_8713.PARAM_COEF := 16#07;
   AI_8713.VALUE_COEF := 0.00617;
   AI_8813.AI_CODE := 16#8813;
   AI_8813.___________0020_0 := false;
   AI_8813.___________0010_2 := false;
   AI_8813.RAW_MIN := -6000;
   AI_8813.RAW_MAX := 13000;
   AI_8813.RAW_NAME := 'Thermal Resistance - 3-wire (Ni500 climate - 618)';
   AI_8813.___________0030_1 := false;
   AI_8813.___________0030_2 := false;
   AI_8813.PARAM_TYPE := 16#08;
   AI_8813.PARAM_RANGE := 16#13;
   AI_8813.PARAM_COEF := 16#08;
   AI_8813.VALUE_COEF := 0.00618;
   AI_8913.AI_CODE := 16#8913;
   AI_8913.___________0020_0 := false;
   AI_8913.___________0010_2 := false;
   AI_8913.RAW_MIN := -6000;
   AI_8913.RAW_MAX := 13000;
   AI_8913.RAW_NAME := 'Thermal Resistance - 3-wire (Ni500 climate - 672)';
   AI_8913.___________0030_1 := false;
   AI_8913.___________0030_2 := false;
   AI_8913.PARAM_TYPE := 16#08;
   AI_8913.PARAM_RANGE := 16#13;
   AI_8913.PARAM_COEF := 16#09;
   AI_8913.VALUE_COEF := 0.00672;
   AI_8712.AI_CODE := 16#8712;
   AI_8712.___________0020_0 := false;
   AI_8712.___________0010_2 := false;
   AI_8712.RAW_MIN := -600;
   AI_8712.RAW_MAX := 1800;
   AI_8712.RAW_NAME := 'Thermal Resistance - 3-wire (Ni500 standard - 617)';
   AI_8712.___________0030_1 := false;
   AI_8712.___________0030_2 := false;
   AI_8712.PARAM_TYPE := 16#08;
   AI_8712.PARAM_RANGE := 16#12;
   AI_8712.PARAM_COEF := 16#07;
   AI_8712.VALUE_COEF := 0.00617;
   AI_8812.AI_CODE := 16#8812;
   AI_8812.___________0020_0 := false;
   AI_8812.___________0010_2 := false;
   AI_8812.RAW_MIN := -600;
   AI_8812.RAW_MAX := 2500;
   AI_8812.RAW_NAME := 'Thermal Resistance - 3-wire (Ni500 standard - 618)';
   AI_8812.___________0030_1 := false;
   AI_8812.___________0030_2 := false;
   AI_8812.PARAM_TYPE := 16#08;
   AI_8812.PARAM_RANGE := 16#12;
   AI_8812.PARAM_COEF := 16#08;
   AI_8812.VALUE_COEF := 0.00618;
   AI_8912.AI_CODE := 16#8912;
   AI_8912.___________0020_0 := false;
   AI_8912.___________0010_2 := false;
   AI_8912.RAW_MIN := -600;
   AI_8912.RAW_MAX := 2500;
   AI_8912.RAW_NAME := 'Thermal Resistance - 3-wire (Ni500 standard - 672)';
   AI_8912.___________0030_1 := false;
   AI_8912.___________0030_2 := false;
   AI_8912.PARAM_TYPE := 16#08;
   AI_8912.PARAM_RANGE := 16#12;
   AI_8912.PARAM_COEF := 16#09;
   AI_8912.VALUE_COEF := 0.00672;
   AI_870A.AI_CODE := 16#870A;
   AI_870A.___________0020_0 := false;
   AI_870A.___________0010_2 := false;
   AI_870A.RAW_MIN := -6000;
   AI_870A.RAW_MAX := 13000;
   AI_870A.RAW_NAME := 'Thermal Resistance - 3-wire (Ni1000 climate - 617)';
   AI_870A.___________0030_1 := false;
   AI_870A.___________0030_2 := false;
   AI_870A.PARAM_TYPE := 16#08;
   AI_870A.PARAM_RANGE := 16#0A;
   AI_870A.PARAM_COEF := 16#07;
   AI_870A.VALUE_COEF := 0.00617;
   AI_880A.AI_CODE := 16#880A;
   AI_880A.___________0020_0 := false;
   AI_880A.___________0010_2 := false;
   AI_880A.RAW_MIN := -6000;
   AI_880A.RAW_MAX := 13000;
   AI_880A.RAW_NAME := 'Thermal Resistance - 3-wire (Ni1000 climate - 618)';
   AI_880A.___________0030_1 := false;
   AI_880A.___________0030_2 := false;
   AI_880A.PARAM_TYPE := 16#08;
   AI_880A.PARAM_RANGE := 16#0A;
   AI_880A.PARAM_COEF := 16#08;
   AI_880A.VALUE_COEF := 0.00618;
   AI_890A.AI_CODE := 16#890A;
   AI_890A.___________0020_0 := false;
   AI_890A.___________0010_2 := false;
   AI_890A.RAW_MIN := -6000;
   AI_890A.RAW_MAX := 13000;
   AI_890A.RAW_NAME := 'Thermal Resistance - 3-wire (Ni1000 climate - 672)';
   AI_890A.___________0030_1 := false;
   AI_890A.___________0030_2 := false;
   AI_890A.PARAM_TYPE := 16#08;
   AI_890A.PARAM_RANGE := 16#0A;
   AI_890A.PARAM_COEF := 16#09;
   AI_890A.VALUE_COEF := 0.00672;
   AI_8706.AI_CODE := 16#8706;
   AI_8706.___________0020_0 := false;
   AI_8706.___________0010_2 := false;
   AI_8706.RAW_MIN := -600;
   AI_8706.RAW_MAX := 1800;
   AI_8706.RAW_NAME := 'Thermal Resistance - 3-wire (Ni1000 standard - 617)';
   AI_8706.___________0030_1 := false;
   AI_8706.___________0030_2 := false;
   AI_8706.PARAM_TYPE := 16#08;
   AI_8706.PARAM_RANGE := 16#06;
   AI_8706.PARAM_COEF := 16#07;
   AI_8706.VALUE_COEF := 0.00617;
   AI_8806.AI_CODE := 16#8806;
   AI_8806.___________0020_0 := false;
   AI_8806.___________0010_2 := false;
   AI_8806.RAW_MIN := -600;
   AI_8806.RAW_MAX := 2500;
   AI_8806.RAW_NAME := 'Thermal Resistance - 3-wire (Ni1000 standard - 618)';
   AI_8806.___________0030_1 := false;
   AI_8806.___________0030_2 := false;
   AI_8806.PARAM_TYPE := 16#08;
   AI_8806.PARAM_RANGE := 16#06;
   AI_8806.PARAM_COEF := 16#08;
   AI_8806.VALUE_COEF := 0.00618;
   AI_8906.AI_CODE := 16#8906;
   AI_8906.___________0020_0 := false;
   AI_8906.___________0010_2 := false;
   AI_8906.RAW_MIN := -600;
   AI_8906.RAW_MAX := 2500;
   AI_8906.RAW_NAME := 'Thermal Resistance - 3-wire (Ni1000 standard - 672)';
   AI_8906.___________0030_1 := false;
   AI_8906.___________0030_2 := false;
   AI_8906.PARAM_TYPE := 16#08;
   AI_8906.PARAM_RANGE := 16#06;
   AI_8906.PARAM_COEF := 16#09;
   AI_8906.VALUE_COEF := 0.00672;
   AI_8015.AI_CODE := 16#8015;
   AI_8015.___________0020_0 := false;
   AI_8015.___________0010_2 := false;
   AI_8015.RAW_MIN := -12000;
   AI_8015.RAW_MAX := 13000;
   AI_8015.RAW_NAME := 'Thermal Resistance - 3-wire (Pt10 climate - 3851)';
   AI_8015.___________0030_1 := false;
   AI_8015.___________0030_2 := false;
   AI_8015.PARAM_TYPE := 16#08;
   AI_8015.PARAM_RANGE := 16#15;
   AI_8015.PARAM_COEF := 16#00;
   AI_8015.VALUE_COEF := 0.003851;
   AI_8215.AI_CODE := 16#8215;
   AI_8215.___________0020_0 := false;
   AI_8215.___________0010_2 := false;
   AI_8215.RAW_MIN := -12000;
   AI_8215.RAW_MAX := 13000;
   AI_8215.RAW_NAME := 'Thermal Resistance - 3-wire (Pt10 climate - 3902)';
   AI_8215.___________0030_1 := false;
   AI_8215.___________0030_2 := false;
   AI_8215.PARAM_TYPE := 16#08;
   AI_8215.PARAM_RANGE := 16#15;
   AI_8215.PARAM_COEF := 16#02;
   AI_8215.VALUE_COEF := 0.003902;
   AI_8515.AI_CODE := 16#8515;
   AI_8515.___________0020_0 := false;
   AI_8515.___________0010_2 := false;
   AI_8515.RAW_MIN := -12000;
   AI_8515.RAW_MAX := 13000;
   AI_8515.RAW_NAME := 'Thermal Resistance - 3-wire (Pt10 climate - 391)';
   AI_8515.___________0030_1 := false;
   AI_8515.___________0030_2 := false;
   AI_8515.PARAM_TYPE := 16#08;
   AI_8515.PARAM_RANGE := 16#15;
   AI_8515.PARAM_COEF := 16#05;
   AI_8515.VALUE_COEF := 0.00391;
   AI_8115.AI_CODE := 16#8115;
   AI_8115.___________0020_0 := false;
   AI_8115.___________0010_2 := false;
   AI_8115.RAW_MIN := -12000;
   AI_8115.RAW_MAX := 13000;
   AI_8115.RAW_NAME := 'Thermal Resistance - 3-wire (Pt10 climate - 3916)';
   AI_8115.___________0030_1 := false;
   AI_8115.___________0030_2 := false;
   AI_8115.PARAM_TYPE := 16#08;
   AI_8115.PARAM_RANGE := 16#15;
   AI_8115.PARAM_COEF := 16#01;
   AI_8115.VALUE_COEF := 0.003916;
   AI_8315.AI_CODE := 16#8315;
   AI_8315.___________0020_0 := false;
   AI_8315.___________0010_2 := false;
   AI_8315.RAW_MIN := -12000;
   AI_8315.RAW_MAX := 13000;
   AI_8315.RAW_NAME := 'Thermal Resistance - 3-wire (Pt10 climate - 392)';
   AI_8315.___________0030_1 := false;
   AI_8315.___________0030_2 := false;
   AI_8315.PARAM_TYPE := 16#08;
   AI_8315.PARAM_RANGE := 16#15;
   AI_8315.PARAM_COEF := 16#03;
   AI_8315.VALUE_COEF := 0.00392;
   AI_8014.AI_CODE := 16#8014;
   AI_8014.___________0020_0 := false;
   AI_8014.___________0010_2 := false;
   AI_8014.RAW_MIN := -2000;
   AI_8014.RAW_MAX := 8500;
   AI_8014.RAW_NAME := 'Thermal Resistance - 3-wire (Pt10 standard - 3851)';
   AI_8014.___________0030_1 := false;
   AI_8014.___________0030_2 := false;
   AI_8014.PARAM_TYPE := 16#08;
   AI_8014.PARAM_RANGE := 16#14;
   AI_8014.PARAM_COEF := 16#00;
   AI_8014.VALUE_COEF := 0.003851;
   AI_8214.AI_CODE := 16#8214;
   AI_8214.___________0020_0 := false;
   AI_8214.___________0010_2 := false;
   AI_8214.RAW_MIN := -2000;
   AI_8214.RAW_MAX := 8500;
   AI_8214.RAW_NAME := 'Thermal Resistance - 3-wire (Pt10 standard - 3902)';
   AI_8214.___________0030_1 := false;
   AI_8214.___________0030_2 := false;
   AI_8214.PARAM_TYPE := 16#08;
   AI_8214.PARAM_RANGE := 16#14;
   AI_8214.PARAM_COEF := 16#02;
   AI_8214.VALUE_COEF := 0.003902;
   AI_8514.AI_CODE := 16#8514;
   AI_8514.___________0020_0 := false;
   AI_8514.___________0010_2 := false;
   AI_8514.RAW_MIN := -2000;
   AI_8514.RAW_MAX := 8500;
   AI_8514.RAW_NAME := 'Thermal Resistance - 3-wire (Pt10 standard - 391)';
   AI_8514.___________0030_1 := false;
   AI_8514.___________0030_2 := false;
   AI_8514.PARAM_TYPE := 16#08;
   AI_8514.PARAM_RANGE := 16#14;
   AI_8514.PARAM_COEF := 16#05;
   AI_8514.VALUE_COEF := 0.00391;
   AI_8114.AI_CODE := 16#8114;
   AI_8114.___________0020_0 := false;
   AI_8114.___________0010_2 := false;
   AI_8114.RAW_MIN := -2000;
   AI_8114.RAW_MAX := 8500;
   AI_8114.RAW_NAME := 'Thermal Resistance - 3-wire (Pt10 standard - 3916)';
   AI_8114.___________0030_1 := false;
   AI_8114.___________0030_2 := false;
   AI_8114.PARAM_TYPE := 16#08;
   AI_8114.PARAM_RANGE := 16#14;
   AI_8114.PARAM_COEF := 16#01;
   AI_8114.VALUE_COEF := 0.003916;
   AI_8314.AI_CODE := 16#8314;
   AI_8314.___________0020_0 := false;
   AI_8314.___________0010_2 := false;
   AI_8314.RAW_MIN := -2000;
   AI_8314.RAW_MAX := 8500;
   AI_8314.RAW_NAME := 'Thermal Resistance - 3-wire (Pt10 standard - 392)';
   AI_8314.___________0030_1 := false;
   AI_8314.___________0030_2 := false;
   AI_8314.PARAM_TYPE := 16#08;
   AI_8314.PARAM_RANGE := 16#14;
   AI_8314.PARAM_COEF := 16#03;
   AI_8314.VALUE_COEF := 0.00392;
   AI_8017.AI_CODE := 16#8017;
   AI_8017.___________0020_0 := false;
   AI_8017.___________0010_2 := false;
   AI_8017.RAW_MIN := -12000;
   AI_8017.RAW_MAX := 13000;
   AI_8017.RAW_NAME := 'Thermal Resistance - 3-wire (Pt50 climate - 3851)';
   AI_8017.___________0030_1 := false;
   AI_8017.___________0030_2 := false;
   AI_8017.PARAM_TYPE := 16#08;
   AI_8017.PARAM_RANGE := 16#17;
   AI_8017.PARAM_COEF := 16#00;
   AI_8017.VALUE_COEF := 0.003851;
   AI_8217.AI_CODE := 16#8217;
   AI_8217.___________0020_0 := false;
   AI_8217.___________0010_2 := false;
   AI_8217.RAW_MIN := -12000;
   AI_8217.RAW_MAX := 13000;
   AI_8217.RAW_NAME := 'Thermal Resistance - 3-wire (Pt50 climate - 3902)';
   AI_8217.___________0030_1 := false;
   AI_8217.___________0030_2 := false;
   AI_8217.PARAM_TYPE := 16#08;
   AI_8217.PARAM_RANGE := 16#17;
   AI_8217.PARAM_COEF := 16#02;
   AI_8217.VALUE_COEF := 0.003902;
   AI_8517.AI_CODE := 16#8517;
   AI_8517.___________0020_0 := false;
   AI_8517.___________0010_2 := false;
   AI_8517.RAW_MIN := -12000;
   AI_8517.RAW_MAX := 13000;
   AI_8517.RAW_NAME := 'Thermal Resistance - 3-wire (Pt50 climate - 391)';
   AI_8517.___________0030_1 := false;
   AI_8517.___________0030_2 := false;
   AI_8517.PARAM_TYPE := 16#08;
   AI_8517.PARAM_RANGE := 16#17;
   AI_8517.PARAM_COEF := 16#05;
   AI_8517.VALUE_COEF := 0.00391;
   AI_8117.AI_CODE := 16#8117;
   AI_8117.___________0020_0 := false;
   AI_8117.___________0010_2 := false;
   AI_8117.RAW_MIN := -12000;
   AI_8117.RAW_MAX := 13000;
   AI_8117.RAW_NAME := 'Thermal Resistance - 3-wire (Pt50 climate - 3916)';
   AI_8117.___________0030_1 := false;
   AI_8117.___________0030_2 := false;
   AI_8117.PARAM_TYPE := 16#08;
   AI_8117.PARAM_RANGE := 16#17;
   AI_8117.PARAM_COEF := 16#01;
   AI_8117.VALUE_COEF := 0.003916;
   AI_8317.AI_CODE := 16#8317;
   AI_8317.___________0020_0 := false;
   AI_8317.___________0010_2 := false;
   AI_8317.RAW_MIN := -12000;
   AI_8317.RAW_MAX := 13000;
   AI_8317.RAW_NAME := 'Thermal Resistance - 3-wire (Pt50 climate - 392)';
   AI_8317.___________0030_1 := false;
   AI_8317.___________0030_2 := false;
   AI_8317.PARAM_TYPE := 16#08;
   AI_8317.PARAM_RANGE := 16#17;
   AI_8317.PARAM_COEF := 16#03;
   AI_8317.VALUE_COEF := 0.00392;
   AI_8016.AI_CODE := 16#8016;
   AI_8016.___________0020_0 := false;
   AI_8016.___________0010_2 := false;
   AI_8016.RAW_MIN := -2000;
   AI_8016.RAW_MAX := 8500;
   AI_8016.RAW_NAME := 'Thermal Resistance - 3-wire (Pt50 standard - 3851)';
   AI_8016.___________0030_1 := false;
   AI_8016.___________0030_2 := false;
   AI_8016.PARAM_TYPE := 16#08;
   AI_8016.PARAM_RANGE := 16#16;
   AI_8016.PARAM_COEF := 16#00;
   AI_8016.VALUE_COEF := 0.003851;
   AI_8216.AI_CODE := 16#8216;
   AI_8216.___________0020_0 := false;
   AI_8216.___________0010_2 := false;
   AI_8216.RAW_MIN := -2000;
   AI_8216.RAW_MAX := 8500;
   AI_8216.RAW_NAME := 'Thermal Resistance - 3-wire (Pt50 standard - 3902)';
   AI_8216.___________0030_1 := false;
   AI_8216.___________0030_2 := false;
   AI_8216.PARAM_TYPE := 16#08;
   AI_8216.PARAM_RANGE := 16#16;
   AI_8216.PARAM_COEF := 16#02;
   AI_8216.VALUE_COEF := 0.003902;
   AI_8516.AI_CODE := 16#8516;
   AI_8516.___________0020_0 := false;
   AI_8516.___________0010_2 := false;
   AI_8516.RAW_MIN := -2000;
   AI_8516.RAW_MAX := 8500;
   AI_8516.RAW_NAME := 'Thermal Resistance - 3-wire (Pt50 standard - 391)';
   AI_8516.___________0030_1 := false;
   AI_8516.___________0030_2 := false;
   AI_8516.PARAM_TYPE := 16#08;
   AI_8516.PARAM_RANGE := 16#16;
   AI_8516.PARAM_COEF := 16#05;
   AI_8516.VALUE_COEF := 0.00391;
   AI_8116.AI_CODE := 16#8116;
   AI_8116.___________0020_0 := false;
   AI_8116.___________0010_2 := false;
   AI_8116.RAW_MIN := -2000;
   AI_8116.RAW_MAX := 8500;
   AI_8116.RAW_NAME := 'Thermal Resistance - 3-wire (Pt50 standard - 3916)';
   AI_8116.___________0030_1 := false;
   AI_8116.___________0030_2 := false;
   AI_8116.PARAM_TYPE := 16#08;
   AI_8116.PARAM_RANGE := 16#16;
   AI_8116.PARAM_COEF := 16#01;
   AI_8116.VALUE_COEF := 0.003916;
   AI_8316.AI_CODE := 16#8316;
   AI_8316.___________0020_0 := false;
   AI_8316.___________0010_2 := false;
   AI_8316.RAW_MIN := -2000;
   AI_8316.RAW_MAX := 8500;
   AI_8316.RAW_NAME := 'Thermal Resistance - 3-wire (Pt50 standard - 392)';
   AI_8316.___________0030_1 := false;
   AI_8316.___________0030_2 := false;
   AI_8316.PARAM_TYPE := 16#08;
   AI_8316.PARAM_RANGE := 16#16;
   AI_8316.PARAM_COEF := 16#03;
   AI_8316.VALUE_COEF := 0.00392;
   AI_8000.AI_CODE := 16#8000;
   AI_8000.___________0020_0 := false;
   AI_8000.___________0010_2 := false;
   AI_8000.RAW_MIN := -12000;
   AI_8000.RAW_MAX := 13000;
   AI_8000.RAW_NAME := 'Thermal Resistance - 3-wire (Pt100 climate - 3851)';
   AI_8000.___________0030_1 := false;
   AI_8000.___________0030_2 := false;
   AI_8000.PARAM_TYPE := 16#08;
   AI_8000.PARAM_RANGE := 16#00;
   AI_8000.PARAM_COEF := 16#00;
   AI_8000.VALUE_COEF := 0.003851;
   AI_8200.AI_CODE := 16#8200;
   AI_8200.___________0020_0 := false;
   AI_8200.___________0010_2 := false;
   AI_8200.RAW_MIN := -12000;
   AI_8200.RAW_MAX := 13000;
   AI_8200.RAW_NAME := 'Thermal Resistance - 3-wire (Pt100 climate - 3902)';
   AI_8200.___________0030_1 := false;
   AI_8200.___________0030_2 := false;
   AI_8200.PARAM_TYPE := 16#08;
   AI_8200.PARAM_RANGE := 16#00;
   AI_8200.PARAM_COEF := 16#02;
   AI_8200.VALUE_COEF := 0.003902;
   AI_8500.AI_CODE := 16#8500;
   AI_8500.___________0020_0 := false;
   AI_8500.___________0010_2 := false;
   AI_8500.RAW_MIN := -12000;
   AI_8500.RAW_MAX := 13000;
   AI_8500.RAW_NAME := 'Thermal Resistance - 3-wire (Pt100 climate - 391)';
   AI_8500.___________0030_1 := false;
   AI_8500.___________0030_2 := false;
   AI_8500.PARAM_TYPE := 16#08;
   AI_8500.PARAM_RANGE := 16#00;
   AI_8500.PARAM_COEF := 16#05;
   AI_8500.VALUE_COEF := 0.00391;
   AI_8100.AI_CODE := 16#8100;
   AI_8100.___________0020_0 := false;
   AI_8100.___________0010_2 := false;
   AI_8100.RAW_MIN := -12000;
   AI_8100.RAW_MAX := 13000;
   AI_8100.RAW_NAME := 'Thermal Resistance - 3-wire (Pt100 climate - 3916)';
   AI_8100.___________0030_1 := false;
   AI_8100.___________0030_2 := false;
   AI_8100.PARAM_TYPE := 16#08;
   AI_8100.PARAM_RANGE := 16#00;
   AI_8100.PARAM_COEF := 16#01;
   AI_8100.VALUE_COEF := 0.003916;
   AI_8300.AI_CODE := 16#8300;
   AI_8300.___________0020_0 := false;
   AI_8300.___________0010_2 := false;
   AI_8300.RAW_MIN := -12000;
   AI_8300.RAW_MAX := 13000;
   AI_8300.RAW_NAME := 'Thermal Resistance - 3-wire (Pt100 climate - 392)';
   AI_8300.___________0030_1 := false;
   AI_8300.___________0030_2 := false;
   AI_8300.PARAM_TYPE := 16#08;
   AI_8300.PARAM_RANGE := 16#00;
   AI_8300.PARAM_COEF := 16#03;
   AI_8300.VALUE_COEF := 0.00392;
   AI_8002.AI_CODE := 16#8002;
   AI_8002.___________0020_0 := false;
   AI_8002.___________0010_2 := false;
   AI_8002.RAW_MIN := -2000;
   AI_8002.RAW_MAX := 8500;
   AI_8002.RAW_NAME := 'Thermal Resistance - 3-wire (Pt100 standard - 3851)';
   AI_8002.___________0030_1 := false;
   AI_8002.___________0030_2 := false;
   AI_8002.PARAM_TYPE := 16#08;
   AI_8002.PARAM_RANGE := 16#02;
   AI_8002.PARAM_COEF := 16#00;
   AI_8002.VALUE_COEF := 0.003851;
   AI_8202.AI_CODE := 16#8202;
   AI_8202.___________0020_0 := false;
   AI_8202.___________0010_2 := false;
   AI_8202.RAW_MIN := -2000;
   AI_8202.RAW_MAX := 8500;
   AI_8202.RAW_NAME := 'Thermal Resistance - 3-wire (Pt100 standard - 3902)';
   AI_8202.___________0030_1 := false;
   AI_8202.___________0030_2 := false;
   AI_8202.PARAM_TYPE := 16#08;
   AI_8202.PARAM_RANGE := 16#02;
   AI_8202.PARAM_COEF := 16#02;
   AI_8202.VALUE_COEF := 0.003902;
   AI_8502.AI_CODE := 16#8502;
   AI_8502.___________0020_0 := false;
   AI_8502.___________0010_2 := false;
   AI_8502.RAW_MIN := -2000;
   AI_8502.RAW_MAX := 8500;
   AI_8502.RAW_NAME := 'Thermal Resistance - 3-wire (Pt100 standard - 391)';
   AI_8502.___________0030_1 := false;
   AI_8502.___________0030_2 := false;
   AI_8502.PARAM_TYPE := 16#08;
   AI_8502.PARAM_RANGE := 16#02;
   AI_8502.PARAM_COEF := 16#05;
   AI_8502.VALUE_COEF := 0.00391;
   AI_8102.AI_CODE := 16#8102;
   AI_8102.___________0020_0 := false;
   AI_8102.___________0010_2 := false;
   AI_8102.RAW_MIN := -2000;
   AI_8102.RAW_MAX := 8500;
   AI_8102.RAW_NAME := 'Thermal Resistance - 3-wire (Pt100 standard - 3916)';
   AI_8102.___________0030_1 := false;
   AI_8102.___________0030_2 := false;
   AI_8102.PARAM_TYPE := 16#08;
   AI_8102.PARAM_RANGE := 16#02;
   AI_8102.PARAM_COEF := 16#01;
   AI_8102.VALUE_COEF := 0.003916;
   AI_8302.AI_CODE := 16#8302;
   AI_8302.___________0020_0 := false;
   AI_8302.___________0010_2 := false;
   AI_8302.RAW_MIN := -2000;
   AI_8302.RAW_MAX := 8500;
   AI_8302.RAW_NAME := 'Thermal Resistance - 3-wire (Pt100 standard - 392)';
   AI_8302.___________0030_1 := false;
   AI_8302.___________0030_2 := false;
   AI_8302.PARAM_TYPE := 16#08;
   AI_8302.PARAM_RANGE := 16#02;
   AI_8302.PARAM_COEF := 16#03;
   AI_8302.VALUE_COEF := 0.00392;
   AI_8007.AI_CODE := 16#8007;
   AI_8007.___________0020_0 := false;
   AI_8007.___________0010_2 := false;
   AI_8007.RAW_MIN := -12000;
   AI_8007.RAW_MAX := 13000;
   AI_8007.RAW_NAME := 'Thermal Resistance - 3-wire (Pt200 climate - 3851)';
   AI_8007.___________0030_1 := false;
   AI_8007.___________0030_2 := false;
   AI_8007.PARAM_TYPE := 16#08;
   AI_8007.PARAM_RANGE := 16#07;
   AI_8007.PARAM_COEF := 16#00;
   AI_8007.VALUE_COEF := 0.003851;
   AI_8207.AI_CODE := 16#8207;
   AI_8207.___________0020_0 := false;
   AI_8207.___________0010_2 := false;
   AI_8207.RAW_MIN := -12000;
   AI_8207.RAW_MAX := 13000;
   AI_8207.RAW_NAME := 'Thermal Resistance - 3-wire (Pt200 climate - 3902)';
   AI_8207.___________0030_1 := false;
   AI_8207.___________0030_2 := false;
   AI_8207.PARAM_TYPE := 16#08;
   AI_8207.PARAM_RANGE := 16#07;
   AI_8207.PARAM_COEF := 16#02;
   AI_8207.VALUE_COEF := 0.003902;
   AI_8507.AI_CODE := 16#8507;
   AI_8507.___________0020_0 := false;
   AI_8507.___________0010_2 := false;
   AI_8507.RAW_MIN := -12000;
   AI_8507.RAW_MAX := 13000;
   AI_8507.RAW_NAME := 'Thermal Resistance - 3-wire (Pt200 climate - 391)';
   AI_8507.___________0030_1 := false;
   AI_8507.___________0030_2 := false;
   AI_8507.PARAM_TYPE := 16#08;
   AI_8507.PARAM_RANGE := 16#07;
   AI_8507.PARAM_COEF := 16#05;
   AI_8507.VALUE_COEF := 0.00391;
   AI_8107.AI_CODE := 16#8107;
   AI_8107.___________0020_0 := false;
   AI_8107.___________0010_2 := false;
   AI_8107.RAW_MIN := -12000;
   AI_8107.RAW_MAX := 13000;
   AI_8107.RAW_NAME := 'Thermal Resistance - 3-wire (Pt200 climate - 3916)';
   AI_8107.___________0030_1 := false;
   AI_8107.___________0030_2 := false;
   AI_8107.PARAM_TYPE := 16#08;
   AI_8107.PARAM_RANGE := 16#07;
   AI_8107.PARAM_COEF := 16#01;
   AI_8107.VALUE_COEF := 0.003916;
   AI_8307.AI_CODE := 16#8307;
   AI_8307.___________0020_0 := false;
   AI_8307.___________0010_2 := false;
   AI_8307.RAW_MIN := -12000;
   AI_8307.RAW_MAX := 13000;
   AI_8307.RAW_NAME := 'Thermal Resistance - 3-wire (Pt200 climate - 392)';
   AI_8307.___________0030_1 := false;
   AI_8307.___________0030_2 := false;
   AI_8307.PARAM_TYPE := 16#08;
   AI_8307.PARAM_RANGE := 16#07;
   AI_8307.PARAM_COEF := 16#03;
   AI_8307.VALUE_COEF := 0.00392;
   AI_800B.AI_CODE := 16#800B;
   AI_800B.___________0020_0 := false;
   AI_800B.___________0010_2 := false;
   AI_800B.RAW_MIN := -2000;
   AI_800B.RAW_MAX := 8500;
   AI_800B.RAW_NAME := 'Thermal Resistance - 3-wire (Pt200 standard - 3851)';
   AI_800B.___________0030_1 := false;
   AI_800B.___________0030_2 := false;
   AI_800B.PARAM_TYPE := 16#08;
   AI_800B.PARAM_RANGE := 16#0B;
   AI_800B.PARAM_COEF := 16#00;
   AI_800B.VALUE_COEF := 0.003851;
   AI_820B.AI_CODE := 16#820B;
   AI_820B.___________0020_0 := false;
   AI_820B.___________0010_2 := false;
   AI_820B.RAW_MIN := -2000;
   AI_820B.RAW_MAX := 8500;
   AI_820B.RAW_NAME := 'Thermal Resistance - 3-wire (Pt200 standard - 3902)';
   AI_820B.___________0030_1 := false;
   AI_820B.___________0030_2 := false;
   AI_820B.PARAM_TYPE := 16#08;
   AI_820B.PARAM_RANGE := 16#0B;
   AI_820B.PARAM_COEF := 16#02;
   AI_820B.VALUE_COEF := 0.003902;
   AI_850B.AI_CODE := 16#850B;
   AI_850B.___________0020_0 := false;
   AI_850B.___________0010_2 := false;
   AI_850B.RAW_MIN := -2000;
   AI_850B.RAW_MAX := 8500;
   AI_850B.RAW_NAME := 'Thermal Resistance - 3-wire (Pt200 standard - 391)';
   AI_850B.___________0030_1 := false;
   AI_850B.___________0030_2 := false;
   AI_850B.PARAM_TYPE := 16#08;
   AI_850B.PARAM_RANGE := 16#0B;
   AI_850B.PARAM_COEF := 16#05;
   AI_850B.VALUE_COEF := 0.00391;
   AI_810B.AI_CODE := 16#810B;
   AI_810B.___________0020_0 := false;
   AI_810B.___________0010_2 := false;
   AI_810B.RAW_MIN := -2000;
   AI_810B.RAW_MAX := 8500;
   AI_810B.RAW_NAME := 'Thermal Resistance - 3-wire (Pt200 standard - 3916)';
   AI_810B.___________0030_1 := false;
   AI_810B.___________0030_2 := false;
   AI_810B.PARAM_TYPE := 16#08;
   AI_810B.PARAM_RANGE := 16#0B;
   AI_810B.PARAM_COEF := 16#01;
   AI_810B.VALUE_COEF := 0.003916;
   AI_830B.AI_CODE := 16#830B;
   AI_830B.___________0020_0 := false;
   AI_830B.___________0010_2 := false;
   AI_830B.RAW_MIN := -2000;
   AI_830B.RAW_MAX := 8500;
   AI_830B.RAW_NAME := 'Thermal Resistance - 3-wire (Pt200 standard - 392)';
   AI_830B.___________0030_1 := false;
   AI_830B.___________0030_2 := false;
   AI_830B.PARAM_TYPE := 16#08;
   AI_830B.PARAM_RANGE := 16#0B;
   AI_830B.PARAM_COEF := 16#03;
   AI_830B.VALUE_COEF := 0.00392;
   AI_8008.AI_CODE := 16#8008;
   AI_8008.___________0020_0 := false;
   AI_8008.___________0010_2 := false;
   AI_8008.RAW_MIN := -12000;
   AI_8008.RAW_MAX := 13000;
   AI_8008.RAW_NAME := 'Thermal Resistance - 3-wire (Pt500 climate - 3851)';
   AI_8008.___________0030_1 := false;
   AI_8008.___________0030_2 := false;
   AI_8008.PARAM_TYPE := 16#08;
   AI_8008.PARAM_RANGE := 16#08;
   AI_8008.PARAM_COEF := 16#00;
   AI_8008.VALUE_COEF := 0.003851;
   AI_8208.AI_CODE := 16#8208;
   AI_8208.___________0020_0 := false;
   AI_8208.___________0010_2 := false;
   AI_8208.RAW_MIN := -12000;
   AI_8208.RAW_MAX := 13000;
   AI_8208.RAW_NAME := 'Thermal Resistance - 3-wire (Pt500 climate - 3902)';
   AI_8208.___________0030_1 := false;
   AI_8208.___________0030_2 := false;
   AI_8208.PARAM_TYPE := 16#08;
   AI_8208.PARAM_RANGE := 16#08;
   AI_8208.PARAM_COEF := 16#02;
   AI_8208.VALUE_COEF := 0.003902;
   AI_8508.AI_CODE := 16#8508;
   AI_8508.___________0020_0 := false;
   AI_8508.___________0010_2 := false;
   AI_8508.RAW_MIN := -12000;
   AI_8508.RAW_MAX := 13000;
   AI_8508.RAW_NAME := 'Thermal Resistance - 3-wire (Pt500 climate - 391)';
   AI_8508.___________0030_1 := false;
   AI_8508.___________0030_2 := false;
   AI_8508.PARAM_TYPE := 16#08;
   AI_8508.PARAM_RANGE := 16#08;
   AI_8508.PARAM_COEF := 16#05;
   AI_8508.VALUE_COEF := 0.00391;
   AI_8108.AI_CODE := 16#8108;
   AI_8108.___________0020_0 := false;
   AI_8108.___________0010_2 := false;
   AI_8108.RAW_MIN := -12000;
   AI_8108.RAW_MAX := 13000;
   AI_8108.RAW_NAME := 'Thermal Resistance - 3-wire (Pt500 climate - 3916)';
   AI_8108.___________0030_1 := false;
   AI_8108.___________0030_2 := false;
   AI_8108.PARAM_TYPE := 16#08;
   AI_8108.PARAM_RANGE := 16#08;
   AI_8108.PARAM_COEF := 16#01;
   AI_8108.VALUE_COEF := 0.003916;
   AI_8308.AI_CODE := 16#8308;
   AI_8308.___________0020_0 := false;
   AI_8308.___________0010_2 := false;
   AI_8308.RAW_MIN := -12000;
   AI_8308.RAW_MAX := 13000;
   AI_8308.RAW_NAME := 'Thermal Resistance - 3-wire (Pt500 climate - 392)';
   AI_8308.___________0030_1 := false;
   AI_8308.___________0030_2 := false;
   AI_8308.PARAM_TYPE := 16#08;
   AI_8308.PARAM_RANGE := 16#08;
   AI_8308.PARAM_COEF := 16#03;
   AI_8308.VALUE_COEF := 0.00392;
   AI_8004.AI_CODE := 16#8004;
   AI_8004.___________0020_0 := false;
   AI_8004.___________0010_2 := false;
   AI_8004.RAW_MIN := -2000;
   AI_8004.RAW_MAX := 8500;
   AI_8004.RAW_NAME := 'Thermal Resistance - 3-wire (Pt500 standard - 3851)';
   AI_8004.___________0030_1 := false;
   AI_8004.___________0030_2 := false;
   AI_8004.PARAM_TYPE := 16#08;
   AI_8004.PARAM_RANGE := 16#04;
   AI_8004.PARAM_COEF := 16#00;
   AI_8004.VALUE_COEF := 0.003851;
   AI_8204.AI_CODE := 16#8204;
   AI_8204.___________0020_0 := false;
   AI_8204.___________0010_2 := false;
   AI_8204.RAW_MIN := -2000;
   AI_8204.RAW_MAX := 8500;
   AI_8204.RAW_NAME := 'Thermal Resistance - 3-wire (Pt500 standard - 3902)';
   AI_8204.___________0030_1 := false;
   AI_8204.___________0030_2 := false;
   AI_8204.PARAM_TYPE := 16#08;
   AI_8204.PARAM_RANGE := 16#04;
   AI_8204.PARAM_COEF := 16#02;
   AI_8204.VALUE_COEF := 0.003902;
   AI_8504.AI_CODE := 16#8504;
   AI_8504.___________0020_0 := false;
   AI_8504.___________0010_2 := false;
   AI_8504.RAW_MIN := -2000;
   AI_8504.RAW_MAX := 8500;
   AI_8504.RAW_NAME := 'Thermal Resistance - 3-wire (Pt500 standard - 391)';
   AI_8504.___________0030_1 := false;
   AI_8504.___________0030_2 := false;
   AI_8504.PARAM_TYPE := 16#08;
   AI_8504.PARAM_RANGE := 16#04;
   AI_8504.PARAM_COEF := 16#05;
   AI_8504.VALUE_COEF := 0.00391;
   AI_8104.AI_CODE := 16#8104;
   AI_8104.___________0020_0 := false;
   AI_8104.___________0010_2 := false;
   AI_8104.RAW_MIN := -2000;
   AI_8104.RAW_MAX := 8500;
   AI_8104.RAW_NAME := 'Thermal Resistance - 3-wire (Pt500 standard - 3916)';
   AI_8104.___________0030_1 := false;
   AI_8104.___________0030_2 := false;
   AI_8104.PARAM_TYPE := 16#08;
   AI_8104.PARAM_RANGE := 16#04;
   AI_8104.PARAM_COEF := 16#01;
   AI_8104.VALUE_COEF := 0.003916;
   AI_8304.AI_CODE := 16#8304;
   AI_8304.___________0020_0 := false;
   AI_8304.___________0010_2 := false;
   AI_8304.RAW_MIN := -2000;
   AI_8304.RAW_MAX := 8500;
   AI_8304.RAW_NAME := 'Thermal Resistance - 3-wire (Pt500 standard - 392)';
   AI_8304.___________0030_1 := false;
   AI_8304.___________0030_2 := false;
   AI_8304.PARAM_TYPE := 16#08;
   AI_8304.PARAM_RANGE := 16#04;
   AI_8304.PARAM_COEF := 16#03;
   AI_8304.VALUE_COEF := 0.00392;
   AI_8009.AI_CODE := 16#8009;
   AI_8009.___________0020_0 := false;
   AI_8009.___________0010_2 := false;
   AI_8009.RAW_MIN := -12000;
   AI_8009.RAW_MAX := 13000;
   AI_8009.RAW_NAME := 'Thermal Resistance - 3-wire (Pt1000 climate - 3851)';
   AI_8009.___________0030_1 := false;
   AI_8009.___________0030_2 := false;
   AI_8009.PARAM_TYPE := 16#08;
   AI_8009.PARAM_RANGE := 16#09;
   AI_8009.PARAM_COEF := 16#00;
   AI_8009.VALUE_COEF := 0.003851;
   AI_8209.AI_CODE := 16#8209;
   AI_8209.___________0020_0 := false;
   AI_8209.___________0010_2 := false;
   AI_8209.RAW_MIN := -12000;
   AI_8209.RAW_MAX := 13000;
   AI_8209.RAW_NAME := 'Thermal Resistance - 3-wire (Pt1000 climate - 3902)';
   AI_8209.___________0030_1 := false;
   AI_8209.___________0030_2 := false;
   AI_8209.PARAM_TYPE := 16#08;
   AI_8209.PARAM_RANGE := 16#09;
   AI_8209.PARAM_COEF := 16#02;
   AI_8209.VALUE_COEF := 0.003902;
   AI_8509.AI_CODE := 16#8509;
   AI_8509.___________0020_0 := false;
   AI_8509.___________0010_2 := false;
   AI_8509.RAW_MIN := -12000;
   AI_8509.RAW_MAX := 13000;
   AI_8509.RAW_NAME := 'Thermal Resistance - 3-wire (Pt1000 climate - 391)';
   AI_8509.___________0030_1 := false;
   AI_8509.___________0030_2 := false;
   AI_8509.PARAM_TYPE := 16#08;
   AI_8509.PARAM_RANGE := 16#09;
   AI_8509.PARAM_COEF := 16#05;
   AI_8509.VALUE_COEF := 0.00391;
   AI_8109.AI_CODE := 16#8109;
   AI_8109.___________0020_0 := false;
   AI_8109.___________0010_2 := false;
   AI_8109.RAW_MIN := -12000;
   AI_8109.RAW_MAX := 13000;
   AI_8109.RAW_NAME := 'Thermal Resistance - 3-wire (Pt1000 climate - 3916)';
   AI_8109.___________0030_1 := false;
   AI_8109.___________0030_2 := false;
   AI_8109.PARAM_TYPE := 16#08;
   AI_8109.PARAM_RANGE := 16#09;
   AI_8109.PARAM_COEF := 16#01;
   AI_8109.VALUE_COEF := 0.003916;
   AI_8309.AI_CODE := 16#8309;
   AI_8309.___________0020_0 := false;
   AI_8309.___________0010_2 := false;
   AI_8309.RAW_MIN := -12000;
   AI_8309.RAW_MAX := 13000;
   AI_8309.RAW_NAME := 'Thermal Resistance - 3-wire (Pt1000 climate - 392)';
   AI_8309.___________0030_1 := false;
   AI_8309.___________0030_2 := false;
   AI_8309.PARAM_TYPE := 16#08;
   AI_8309.PARAM_RANGE := 16#09;
   AI_8309.PARAM_COEF := 16#03;
   AI_8309.VALUE_COEF := 0.00392;
   AI_8005.AI_CODE := 16#8005;
   AI_8005.___________0020_0 := false;
   AI_8005.___________0010_2 := false;
   AI_8005.RAW_MIN := -2000;
   AI_8005.RAW_MAX := 8500;
   AI_8005.RAW_NAME := 'Thermal Resistance - 3-wire (Pt1000 standard - 3851)';
   AI_8005.___________0030_1 := false;
   AI_8005.___________0030_2 := false;
   AI_8005.PARAM_TYPE := 16#08;
   AI_8005.PARAM_RANGE := 16#05;
   AI_8005.PARAM_COEF := 16#00;
   AI_8005.VALUE_COEF := 0.003851;
   AI_8205.AI_CODE := 16#8205;
   AI_8205.___________0020_0 := false;
   AI_8205.___________0010_2 := false;
   AI_8205.RAW_MIN := -2000;
   AI_8205.RAW_MAX := 8500;
   AI_8205.RAW_NAME := 'Thermal Resistance - 3-wire (Pt1000 standard - 3902)';
   AI_8205.___________0030_1 := false;
   AI_8205.___________0030_2 := false;
   AI_8205.PARAM_TYPE := 16#08;
   AI_8205.PARAM_RANGE := 16#05;
   AI_8205.PARAM_COEF := 16#02;
   AI_8205.VALUE_COEF := 0.003902;
   AI_8505.AI_CODE := 16#8505;
   AI_8505.___________0020_0 := false;
   AI_8505.___________0010_2 := false;
   AI_8505.RAW_MIN := -2000;
   AI_8505.RAW_MAX := 8500;
   AI_8505.RAW_NAME := 'Thermal Resistance - 3-wire (Pt1000 standard - 391)';
   AI_8505.___________0030_1 := false;
   AI_8505.___________0030_2 := false;
   AI_8505.PARAM_TYPE := 16#08;
   AI_8505.PARAM_RANGE := 16#05;
   AI_8505.PARAM_COEF := 16#05;
   AI_8505.VALUE_COEF := 0.00391;
   AI_8105.AI_CODE := 16#8105;
   AI_8105.___________0020_0 := false;
   AI_8105.___________0010_2 := false;
   AI_8105.RAW_MIN := -2000;
   AI_8105.RAW_MAX := 8500;
   AI_8105.RAW_NAME := 'Thermal Resistance - 3-wire (Pt1000 standard - 3916)';
   AI_8105.___________0030_1 := false;
   AI_8105.___________0030_2 := false;
   AI_8105.PARAM_TYPE := 16#08;
   AI_8105.PARAM_RANGE := 16#05;
   AI_8105.PARAM_COEF := 16#01;
   AI_8105.VALUE_COEF := 0.003916;
   AI_8305.AI_CODE := 16#8305;
   AI_8305.___________0020_0 := false;
   AI_8305.___________0010_2 := false;
   AI_8305.RAW_MIN := -2000;
   AI_8305.RAW_MAX := 8500;
   AI_8305.RAW_NAME := 'Thermal Resistance - 3-wire (Pt1000 standard - 392)';
   AI_8305.___________0030_1 := false;
   AI_8305.___________0030_2 := false;
   AI_8305.PARAM_TYPE := 16#08;
   AI_8305.PARAM_RANGE := 16#05;
   AI_8305.PARAM_COEF := 16#03;
   AI_8305.VALUE_COEF := 0.00392;
   AI_A000.AI_CODE := 16#A000;
   AI_A000.___________0020_0 := false;
   AI_A000.___________0010_2 := false;
   AI_A000.RAW_MIN := 2500;
   AI_A000.RAW_MAX := 18200;
   AI_A000.RAW_NAME := 'Thermocouple (Type B)';
   AI_A000.___________0030_1 := false;
   AI_A000.___________0030_2 := false;
   AI_A000.PARAM_TYPE := 16#0A;
   AI_A000.PARAM_RANGE := 16#00;
   AI_A000.PARAM_COEF := 16#00;
   AI_A00A.AI_CODE := 16#A00A;
   AI_A00A.___________0020_0 := false;
   AI_A00A.___________0010_2 := false;
   AI_A00A.RAW_MIN := 0;
   AI_A00A.RAW_MAX := 23000;
   AI_A00A.RAW_NAME := 'Thermocouple (Type C)';
   AI_A00A.___________0030_1 := false;
   AI_A00A.___________0030_2 := false;
   AI_A00A.PARAM_TYPE := 16#0A;
   AI_A00A.PARAM_RANGE := 16#0A;
   AI_A00A.PARAM_COEF := 16#00;
   AI_A002.AI_CODE := 16#A002;
   AI_A002.___________0020_0 := false;
   AI_A002.___________0010_2 := false;
   AI_A002.RAW_MIN := -2700;
   AI_A002.RAW_MAX := 10000;
   AI_A002.RAW_NAME := 'Thermocouple (Type E)';
   AI_A002.___________0030_1 := false;
   AI_A002.___________0030_2 := false;
   AI_A002.PARAM_TYPE := 16#0A;
   AI_A002.PARAM_RANGE := 16#02;
   AI_A002.PARAM_COEF := 16#00;
   AI_A005.AI_CODE := 16#A005;
   AI_A005.___________0020_0 := false;
   AI_A005.___________0010_2 := false;
   AI_A005.RAW_MIN := -2100;
   AI_A005.RAW_MAX := 12000;
   AI_A005.RAW_NAME := 'Thermocouple (Type J)';
   AI_A005.___________0030_1 := false;
   AI_A005.___________0030_2 := false;
   AI_A005.PARAM_TYPE := 16#0A;
   AI_A005.PARAM_RANGE := 16#05;
   AI_A005.PARAM_COEF := 16#00;
   AI_A008.AI_CODE := 16#A008;
   AI_A008.___________0020_0 := false;
   AI_A008.___________0010_2 := false;
   AI_A008.RAW_MIN := -2700;
   AI_A008.RAW_MAX := 13720;
   AI_A008.RAW_NAME := 'Thermocouple (Type K)';
   AI_A008.___________0030_1 := false;
   AI_A008.___________0030_2 := false;
   AI_A008.PARAM_TYPE := 16#0A;
   AI_A008.PARAM_RANGE := 16#08;
   AI_A008.PARAM_COEF := 16#00;
   AI_A001.AI_CODE := 16#A001;
   AI_A001.___________0020_0 := false;
   AI_A001.___________0010_2 := false;
   AI_A001.RAW_MIN := -2700;
   AI_A001.RAW_MAX := 13000;
   AI_A001.RAW_NAME := 'Thermocouple (Type N)';
   AI_A001.___________0030_1 := false;
   AI_A001.___________0030_2 := false;
   AI_A001.PARAM_TYPE := 16#0A;
   AI_A001.PARAM_RANGE := 16#01;
   AI_A001.PARAM_COEF := 16#00;
   AI_A003.AI_CODE := 16#A003;
   AI_A003.___________0020_0 := false;
   AI_A003.___________0010_2 := false;
   AI_A003.RAW_MIN := -500;
   AI_A003.RAW_MAX := 17690;
   AI_A003.RAW_NAME := 'Thermocouple (Type R)';
   AI_A003.___________0030_1 := false;
   AI_A003.___________0030_2 := false;
   AI_A003.PARAM_TYPE := 16#0A;
   AI_A003.PARAM_RANGE := 16#03;
   AI_A003.PARAM_COEF := 16#00;
   AI_A004.AI_CODE := 16#A004;
   AI_A004.___________0020_0 := false;
   AI_A004.___________0010_2 := false;
   AI_A004.RAW_MIN := -500;
   AI_A004.RAW_MAX := 17690;
   AI_A004.RAW_NAME := 'Thermocouple (Type S)';
   AI_A004.___________0030_1 := false;
   AI_A004.___________0030_2 := false;
   AI_A004.PARAM_TYPE := 16#0A;
   AI_A004.PARAM_RANGE := 16#04;
   AI_A004.PARAM_COEF := 16#00;
   AI_A007.AI_CODE := 16#A007;
   AI_A007.___________0020_0 := false;
   AI_A007.___________0010_2 := false;
   AI_A007.RAW_MIN := -2700;
   AI_A007.RAW_MAX := 4000;
   AI_A007.RAW_NAME := 'Thermocouple (Type T)';
   AI_A007.___________0030_1 := false;
   AI_A007.___________0030_2 := false;
   AI_A007.PARAM_TYPE := 16#0A;
   AI_A007.PARAM_RANGE := 16#07;
   AI_A007.PARAM_COEF := 16#00;
   AI_A00B.AI_CODE := 16#A00B;
   AI_A00B.___________0020_0 := false;
   AI_A00B.___________0010_2 := false;
   AI_A00B.RAW_MIN := -2000;
   AI_A00B.RAW_MAX := 8000;
   AI_A00B.RAW_NAME := 'Thermocouple (Type TXK/XCL)';
   AI_A00B.___________0030_1 := false;
   AI_A00B.___________0030_2 := false;
   AI_A00B.PARAM_TYPE := 16#0A;
   AI_A00B.PARAM_RANGE := 16#0B;
   AI_A00B.PARAM_COEF := 16#00;
END_DATA_BLOCK
